// TIA Portal V20 export
TYPE "LER_typeEmRelation"
// stored: Access Published, Namespace Unit1
   STRUCT
      em0 { ExternalWritable := 'False'} : "Unit1.typeEm0Standard";
      em1 { ExternalWritable := 'False'} : "Unit1.typeEm1Standard";
      em2 { ExternalWritable := 'False'} : "Unit1.typeEm2Standard";
      em3 { ExternalWritable := 'False'} : "Unit1.typeEm3Standard";
      em4 { ExternalWritable := 'False'} : "Unit1.typeEm4Standard";
      em5 { ExternalWritable := 'False'} : "Unit1.typeEm5Standard";
      em6 { ExternalWritable := 'False'} : "Unit1.typeEm6Standard";
      em7 { ExternalWritable := 'False'} : "Unit1.typeEm7Standard";
   END_STRUCT;
END_TYPE
